FUNCTION_BLOCK TimeBlock (* Basic Function Block Type *)
  (* Standard: 61499-2 *)
  (* Version 0.0, 3/2/2019, vshatrov, nxtControl GmbH, Template *)
  PACKAGE Main;
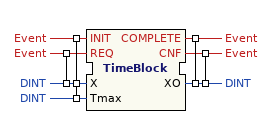
  EVENT_INPUT
    INIT WITH X, Tmax; (* Initialization Request *)
    REQ WITH X; (* Normal Execution Request *)
  END_EVENT
  EVENT_OUTPUT
    COMPLETE WITH XO; (* Initialization Confirm *)
    CNF WITH XO; (* Execution Confirmation *)
  END_EVENT
  VAR_INPUT
    X : DINT; (* Input event qualifier *)
    Tmax : DINT := 20;
  END_VAR
  VAR_OUTPUT
    XO : DINT; (* Output event qualifier *)
  END_VAR
  VAR
    stop : BOOL;
  END_VAR
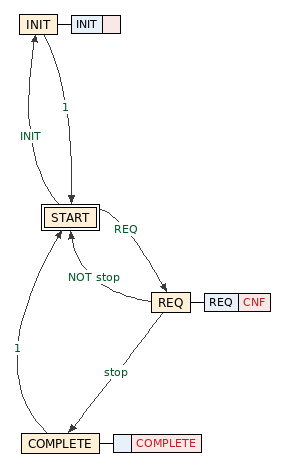
  EC_STATES
    START; (* Initial State *)
    INIT : INIT; (* Initialization *)
    REQ : REQ -> CNF; (* Normal execution *)
    COMPLETE : -> COMPLETE;
  END_STATES
  EC_TRANSITIONS
    START TO INIT := INIT;
    INIT TO START := 1;
    START TO REQ := REQ;
    REQ TO START := NOT stop;
    REQ TO COMPLETE := stop;
    COMPLETE TO START := 1;
  END_TRANSITIONS
  ALGORITHM INIT IN ST: (* Initialization algorithm *)
;
stop := FALSE;
  END_ALGORITHM
  ALGORITHM REQ IN ST: (* Normally executed algorithm *)
;

XO := X + 1;
IF (INVOKEDBY.ts_last - INVOKEDBY.ts_born > Tmax) THEN
	stop := TRUE;
END_IF;
  END_ALGORITHM
END_FUNCTION_BLOCK
